FUNCTION F_CelsiustoFahrenheit : REAL
VAR_INPUT
		fCelsius : REAL;
END_VAR
VAR
END_VAR

F_CelsiustoFahrenheit := fCelsius*1.8 + 32.0;

END_FUNCTION

(* stored: Version 1.1.0.1, ProductVersion 3.1.4024.16
   POU F_CelsiustoFahrenheit: Id {5615a6d7-436e-418e-a2ca-da110f845913}, SpecialFunc None *)
